GLOBALCONSTANTS IG2_Device_Classes (* Industry Group 2 specific device classes (vehicle systems) *)
  (* Standard: 61499-1 *)
  (* Version 1.0, 2026-06-30, Franz Höpfinger, Demmler Andreas Fahrzeugbau *)
  PACKAGE isobus::pgn::const;
  VAR_GLOBAL CONSTANT
    DC_NON_SPECIFIC_SYSTEM : BYTE := 0; (* Device Class / Vehicle System: Non-specific System *)
    DC_TRACTOR : BYTE := 1; (* Device Class / Vehicle System: Tractor *)
    DC_TILLAGE : BYTE := 2; (* Device Class / Vehicle System: Tillage *)
    DC_SECONDARY_TILLAGE : BYTE := 3; (* Device Class / Vehicle System: Secondary Tillage *)
    DC_PLANTERS_SEEDERS : BYTE := 4; (* Device Class / Vehicle System: Planters/Seeders *)
    DC_FERTILIZERS : BYTE := 5; (* Device Class / Vehicle System: Fertilizers *)
    DC_SPRAYERS : BYTE := 6; (* Device Class / Vehicle System: Sprayers *)
    DC_HARVESTERS : BYTE := 7; (* Device Class / Vehicle System: Harvesters *)
    DC_ROOT_HARVESTERS : BYTE := 8; (* Device Class / Vehicle System: Root Harvesters *)
    DC_FORAGE : BYTE := 9; (* Device Class / Vehicle System: Forage *)
    DC_IRRIGATION : BYTE := 10; (* Device Class / Vehicle System: Irrigation *)
    DC_TRANSPORT_TRAILER : BYTE := 11; (* Device Class / Vehicle System: Transport/Trailer *)
    DC_FARM_YARD_OPERATIONS : BYTE := 12; (* Device Class / Vehicle System: Farm Yard Operations *)
    DC_POWERED_AUXILIARY_DEVICES : BYTE := 13; (* Device Class / Vehicle System: Powered Auxiliary Devices *)
    DC_SPECIAL_CROPS : BYTE := 14; (* Device Class / Vehicle System: Special Crops *)
    DC_EARTH_WORK : BYTE := 15; (* Device Class / Vehicle System: Earth Work *)
    DC_SKIDDER : BYTE := 16; (* Device Class / Vehicle System: Skidder *)
    DC_SENSOR_SYSTEMS : BYTE := 17; (* Device Class / Vehicle System: Sensor Systems *)
    DC_TIMBER_HARVESTERS : BYTE := 19; (* Device Class / Vehicle System: Timber Harvesters *)
    DC_FORWARDERS : BYTE := 20; (* Device Class / Vehicle System: Forwarders *)
    DC_TIMBER_LOADERS : BYTE := 21; (* Device Class / Vehicle System: Timber Loaders *)
    DC_TIMBER_PROCESSING_MACHINES : BYTE := 22; (* Device Class / Vehicle System: Timber Processing Machines *)
    DC_MULCHERS : BYTE := 23; (* Device Class / Vehicle System: Mulchers *)
    DC_UTILITY_VEHICLES : BYTE := 24; (* Device Class / Vehicle System: Utility Vehicles *)
    DC_SLURRY_MANURE_APPLICATORS : BYTE := 25; (* Device Class / Vehicle System: Slurry/Manure Applicators *)
    DC_FEEDERS_MIXERS : BYTE := 26; (* Device Class / Vehicle System: Feeders/Mixers *)
    DC_WEEDERS : BYTE := 27; (* Device Class / Vehicle System: Weeders - Non-chemical weed control. The device class Weeders is *)
    DC_TURF_AND_LAWN_CARE_MOWERS : BYTE := 28; (* Device Class / Vehicle System: Turf and Lawn Care Mowers *)
    DC_PRODUCT_MATERIAL_HANDLING : BYTE := 29; (* Device Class / Vehicle System: Product/Material Handling *)
    DC_NOT_AVAILABLE : BYTE := 127; (* Device Class / Vehicle System: Not Available *)
  END_VAR
END_GLOBALCONSTANTS
